{attribute 'linkalways'} 
{attribute 'no_explicit_call' := 'This FB is a CLASS and must be accessed using methods or properties'}
{attribute 'enable_dynamic_creation'}
FUNCTION_BLOCK _ETcVnVectorCompareMethod EXTENDS EnumDatatypeBase
VAR
	localData : ETcVnVectorCompareMethod;
	activeData : REFERENCE TO ETcVnVectorCompareMethod;
	enumBaseDatatype : _DINT(localData);
END_VAR

METHOD PRIVATE AddLocalEnumeration
VAR_INPUT
	Enumeration : T_MAXSTRING;
	Value : ETcVnVectorCompareMethod;
END_VAR
AddEnumeration(Enumeration, Value);
END_METHOD

PROPERTY PUBLIC Address : PVOID
GET
Address := ADR(activeData);
END_GET
END_PROPERTY

METHOD PUBLIC ClearReference
VAR_INPUT
END_VAR
activeData REF= localData;
SetBaseDatatypeReference();
END_METHOD

METHOD PUBLIC Clone : I_Datatype
VAR
    pClone : POINTER TO _ETcVnVectorCompareMethod;
END_VAR
pClone := __NEW(_ETcVnVectorCompareMethod(InitialValue := Value));
Clone := pClone^;
END_METHOD

METHOD FB_init : BOOL
VAR_INPUT
	bInitRetains : BOOL; // if TRUE, the retain variables are initialized (warm start / cold start)
	bInCopyCode : BOOL;  // if TRUE, the instance afterwards gets moved into the copy code (online change)
	InitialValue : ETcVnVectorCompareMethod;
END_VAR
localData := InitialValue;
AddBaseDatatype(enumBaseDatatype);
ClearReference();

AddLocalEnumeration('TCVN_VCM_EUCLIDEAN', ETcVnVectorCompareMethod.TCVN_VCM_EUCLIDEAN);
AddLocalEnumeration('TCVN_VCM_ELEMENTWISE', ETcVnVectorCompareMethod.TCVN_VCM_ELEMENTWISE);
END_METHOD

PROPERTY PUBLIC Identifier : T_MAXSTRING
GET
Identifier := 'ETcVnVectorCompareMethod';
END_GET
END_PROPERTY

METHOD IsEnumeratorValueEqual : BOOL
VAR_INPUT
	Enumerator : I_KeyValueForwardEnumerator;
END_VAR
VAR
	storedValue : ETcVnVectorCompareMethod;
END_VAR
IF NOT Enumerator.TryGet(storedValue) THEN
	RETURN;
END_IF

IsEnumeratorValueEqual := storedValue = activeData;
END_METHOD

METHOD PUBLIC MakeReferenceTo
VAR_INPUT
	ReferenceTarget : REFERENCE TO ETcVnVectorCompareMethod;
END_VAR
activeData REF= ReferenceTarget;
SetBaseDatatypeReference();
END_METHOD

METHOD PROTECTED SetBaseDatatypeReference
VAR_INPUT
END_VAR
enumBaseDatatype.MakeReferenceTo(activeData);
END_METHOD

PROPERTY PUBLIC Size : UDINT
GET
Size := SIZEOF(activeData);
END_GET
END_PROPERTY

METHOD TryMakeReferenceTo : BOOL
VAR_INPUT
	Target : I_Datatype;
END_VAR
VAR
	targetAsEnum : I_EnumDatatype;
	pTargetData : POINTER TO ETcVnVectorCompareMethod;
END_VAR
IF NOT Target.TryResolveAsEnumDatatype(targetAsEnum) THEN
	RETURN;
END_IF

IF targetAsEnum.Identifier <> Identifier THEN
	RETURN;
END_IF

pTargetData := Target.Address;
activeData REF= pTargetData^;
SetBaseDatatypeReference();
TryMakeReferenceTo := TRUE;
END_METHOD

PROPERTY PUBLIC Value : ETcVnVectorCompareMethod
GET
Value := activeData;
END_GET
SET
activeData := Value;
END_SET
END_PROPERTY

END_FUNCTION_BLOCK

(* stored: Version 1.1.0.1, ProductVersion 3.1.4024.12
   POU _ETcVnVectorCompareMethod: Id {99f6ac00-6182-494c-976a-a33e0f494ccf}, SpecialFunc None
   Folder Constructor: Id {c2bcfaf0-e0d6-42ea-a74a-ca6e1c90d593}
   Folder Private: Id {be763214-8164-409c-9a83-5858dff1d8e6}
   Folder Protected: Id {90834b6b-6319-4bec-96fd-f6368f7b332e}
   Method AddLocalEnumeration: Id {79b93fa4-9d2e-4fb4-9224-2ba87381007b}
   Property Address: Id {000e59a3-e92f-4465-887b-f56aae2c8963}
   Get Get: Id {cdfe5058-2ae2-44ec-b046-f73c35d07f12}
   Method ClearReference: Id {b3c269c9-dfa8-4c6d-bbfa-3594ac3473fa}
   Method Clone: Id {810c5579-c221-4351-9232-b862c615aeec}
   Method FB_init: Id {f278d690-bdcf-43da-8858-8186563cf36b}
   Property Identifier: Id {8173252a-1398-4c60-92a4-1c280f520d01}
   Get Get: Id {eaae07d9-888a-4bf8-896b-bfcc61d80cd5}
   Method IsEnumeratorValueEqual: Id {59321a4e-2af1-4427-b5ce-ac1688e01764}
   Method MakeReferenceTo: Id {aac3b1dc-680c-408f-9e84-17f101a11a23}
   Method SetBaseDatatypeReference: Id {c79e160d-6ebf-48db-a078-b3115e78e661}
   Property Size: Id {67c9b334-0d54-4e16-8dc5-69e2627f30b0}
   Get Get: Id {7a73d992-652c-452c-b0fc-0522d633bcbb}
   Method TryMakeReferenceTo: Id {8bafef9c-735b-43bf-8a2b-b817f1c809bc}
   Property Value: Id {b7a98c6d-c4c6-4745-871d-2c1165861bfd}
   Get Get: Id {d559b923-3077-49ab-9164-fcab0398f4b7}
   Set Set: Id {3af0da8a-bd79-4187-90ee-8ec6f830d8ce} *)
